ACTION A502_Suspending_Exit:
{attribute 'hide'}
IF NOT in_bDisableStateMethods THEN
	THIS^.M502_Suspending_Exit();
END_IF
END_ACTION

{attribute 'hide'}
METHOD M500_Suspending_Entry : BOOL
END_METHOD

{attribute 'hide'}
METHOD M501_Suspending : BOOL
VAR_OUTPUT
	(* Move to the Suspended state*)
	bSuspended	: BOOL	:= FALSE;
	(* Move to the Stopping state*)
	bStop		: BOOL	:= FALSE;
	(* Move to the Aborting state*)
	bAbort		: BOOL	:= FALSE;
END_VAR
// Go to suspended state by default
bSuspended := TRUE;
END_METHOD

{attribute 'hide'}
METHOD M502_Suspending_Exit : BOOL
END_METHOD

ACTION A510_Suspended_Entry:
{attribute 'hide'}
sm_enumState := E_PackMLState.Suspended;
sm_bUnsuspend := FALSE;

IF NOT in_bDisableStateMethods THEN
	THIS^.M_LogMessage('Entered $'Suspended$' state.');
	THIS^.M510_Suspended_Entry();
ELSE
	THIS^.M_LogWarning('State methods disabled! Entered $'Suspended$' state. Waiting for transition...');
END_IF
END_ACTION

ACTION A511_Suspended:
{attribute 'hide'}
IF NOT in_bDisableStateMethods THEN
	THIS^.M511_Suspended(
		bUnsuspend => sm_bUnsuspendCmd,
		bStop => sm_bStopCmd,
		bAbort => sm_bAbortCmd);
	IF sm_bAbortCmd THEN
		sm_bAbort := TRUE;
	ELSIF sm_bStopCmd THEN
		sm_bStop := TRUE;
	ELSIF sm_bUnsuspendCmd THEN
		sm_bUnsuspend := TRUE;
	END_IF
END_IF
END_ACTION

ACTION A512_Suspended_Exit:
{attribute 'hide'}
IF NOT in_bDisableStateMethods THEN
	THIS^.M512_Suspended_Exit();
END_IF
END_ACTION

{attribute 'hide'}
METHOD M510_Suspended_Entry : BOOL
END_METHOD

{attribute 'hide'}
METHOD M511_Suspended : BOOL
VAR_OUTPUT
	(* Move to the Unsuspending state*)
	bUnsuspend	: BOOL	:= FALSE;
	(* Move to the Stopping state*)
	bStop		: BOOL	:= FALSE;
	(* Move to the Aborting state*)
	bAbort		: BOOL	:= FALSE;
END_VAR
END_METHOD

{attribute 'hide'}
METHOD M512_Suspended_Exit : BOOL
END_METHOD

ACTION A520_Unsuspending_Entry:
{attribute 'hide'}
sm_enumState := E_PackMLState.Unsuspending;
sm_bUnsuspended := FALSE;

IF NOT in_bDisableStateMethods THEN
	THIS^.M_LogMessage('Entered $'Unsuspending$' state.');
	THIS^.M520_Unsuspending_Entry();
ELSE
	THIS^.M_LogWarning('State methods disabled! Entered $'Unsuspending$' state. Skipping to $'Execute$' state...');
	sm_bUnsuspended := TRUE;
END_IF
END_ACTION

ACTION A521_Unsuspending:
{attribute 'hide'}
IF NOT in_bDisableStateMethods THEN
	THIS^.M521_Unsuspending(
		bUnsuspended => sm_bUnsuspendedCmd,
		bStop => sm_bStopCmd,
		bAbort => sm_bAbortCmd);
	IF sm_bAbortCmd THEN
		sm_bAbort := TRUE;
	ELSIF sm_bStopCmd THEN
		sm_bStop := TRUE;
	ELSIF sm_bUnsuspendedCmd THEN
		sm_bUnsuspended := TRUE;
	END_IF
END_IF
END_ACTION

ACTION A522_Unsuspending_Exit:
{attribute 'hide'}
IF NOT in_bDisableStateMethods THEN
	THIS^.M522_Unsuspending_Exit();
END_IF
END_ACTION

{attribute 'hide'}
METHOD M520_Unsuspending_Entry : BOOL
END_METHOD

{attribute 'hide'}
METHOD M521_Unsuspending : BOOL
VAR_OUTPUT
	(* Move to the Execute state*)
	bUnsuspended	: BOOL	:= FALSE;
	(* Move to the Stopping state*)
	bStop			: BOOL	:= FALSE;
	(* Move to the Aborting state*)
	bAbort			: BOOL	:= FALSE;
END_VAR
// Move to the execute state by default
bUnsuspended := TRUE;
END_METHOD

{attribute 'hide'}
METHOD M522_Unsuspending_Exit : BOOL
END_METHOD

ACTION A_StateMachine:
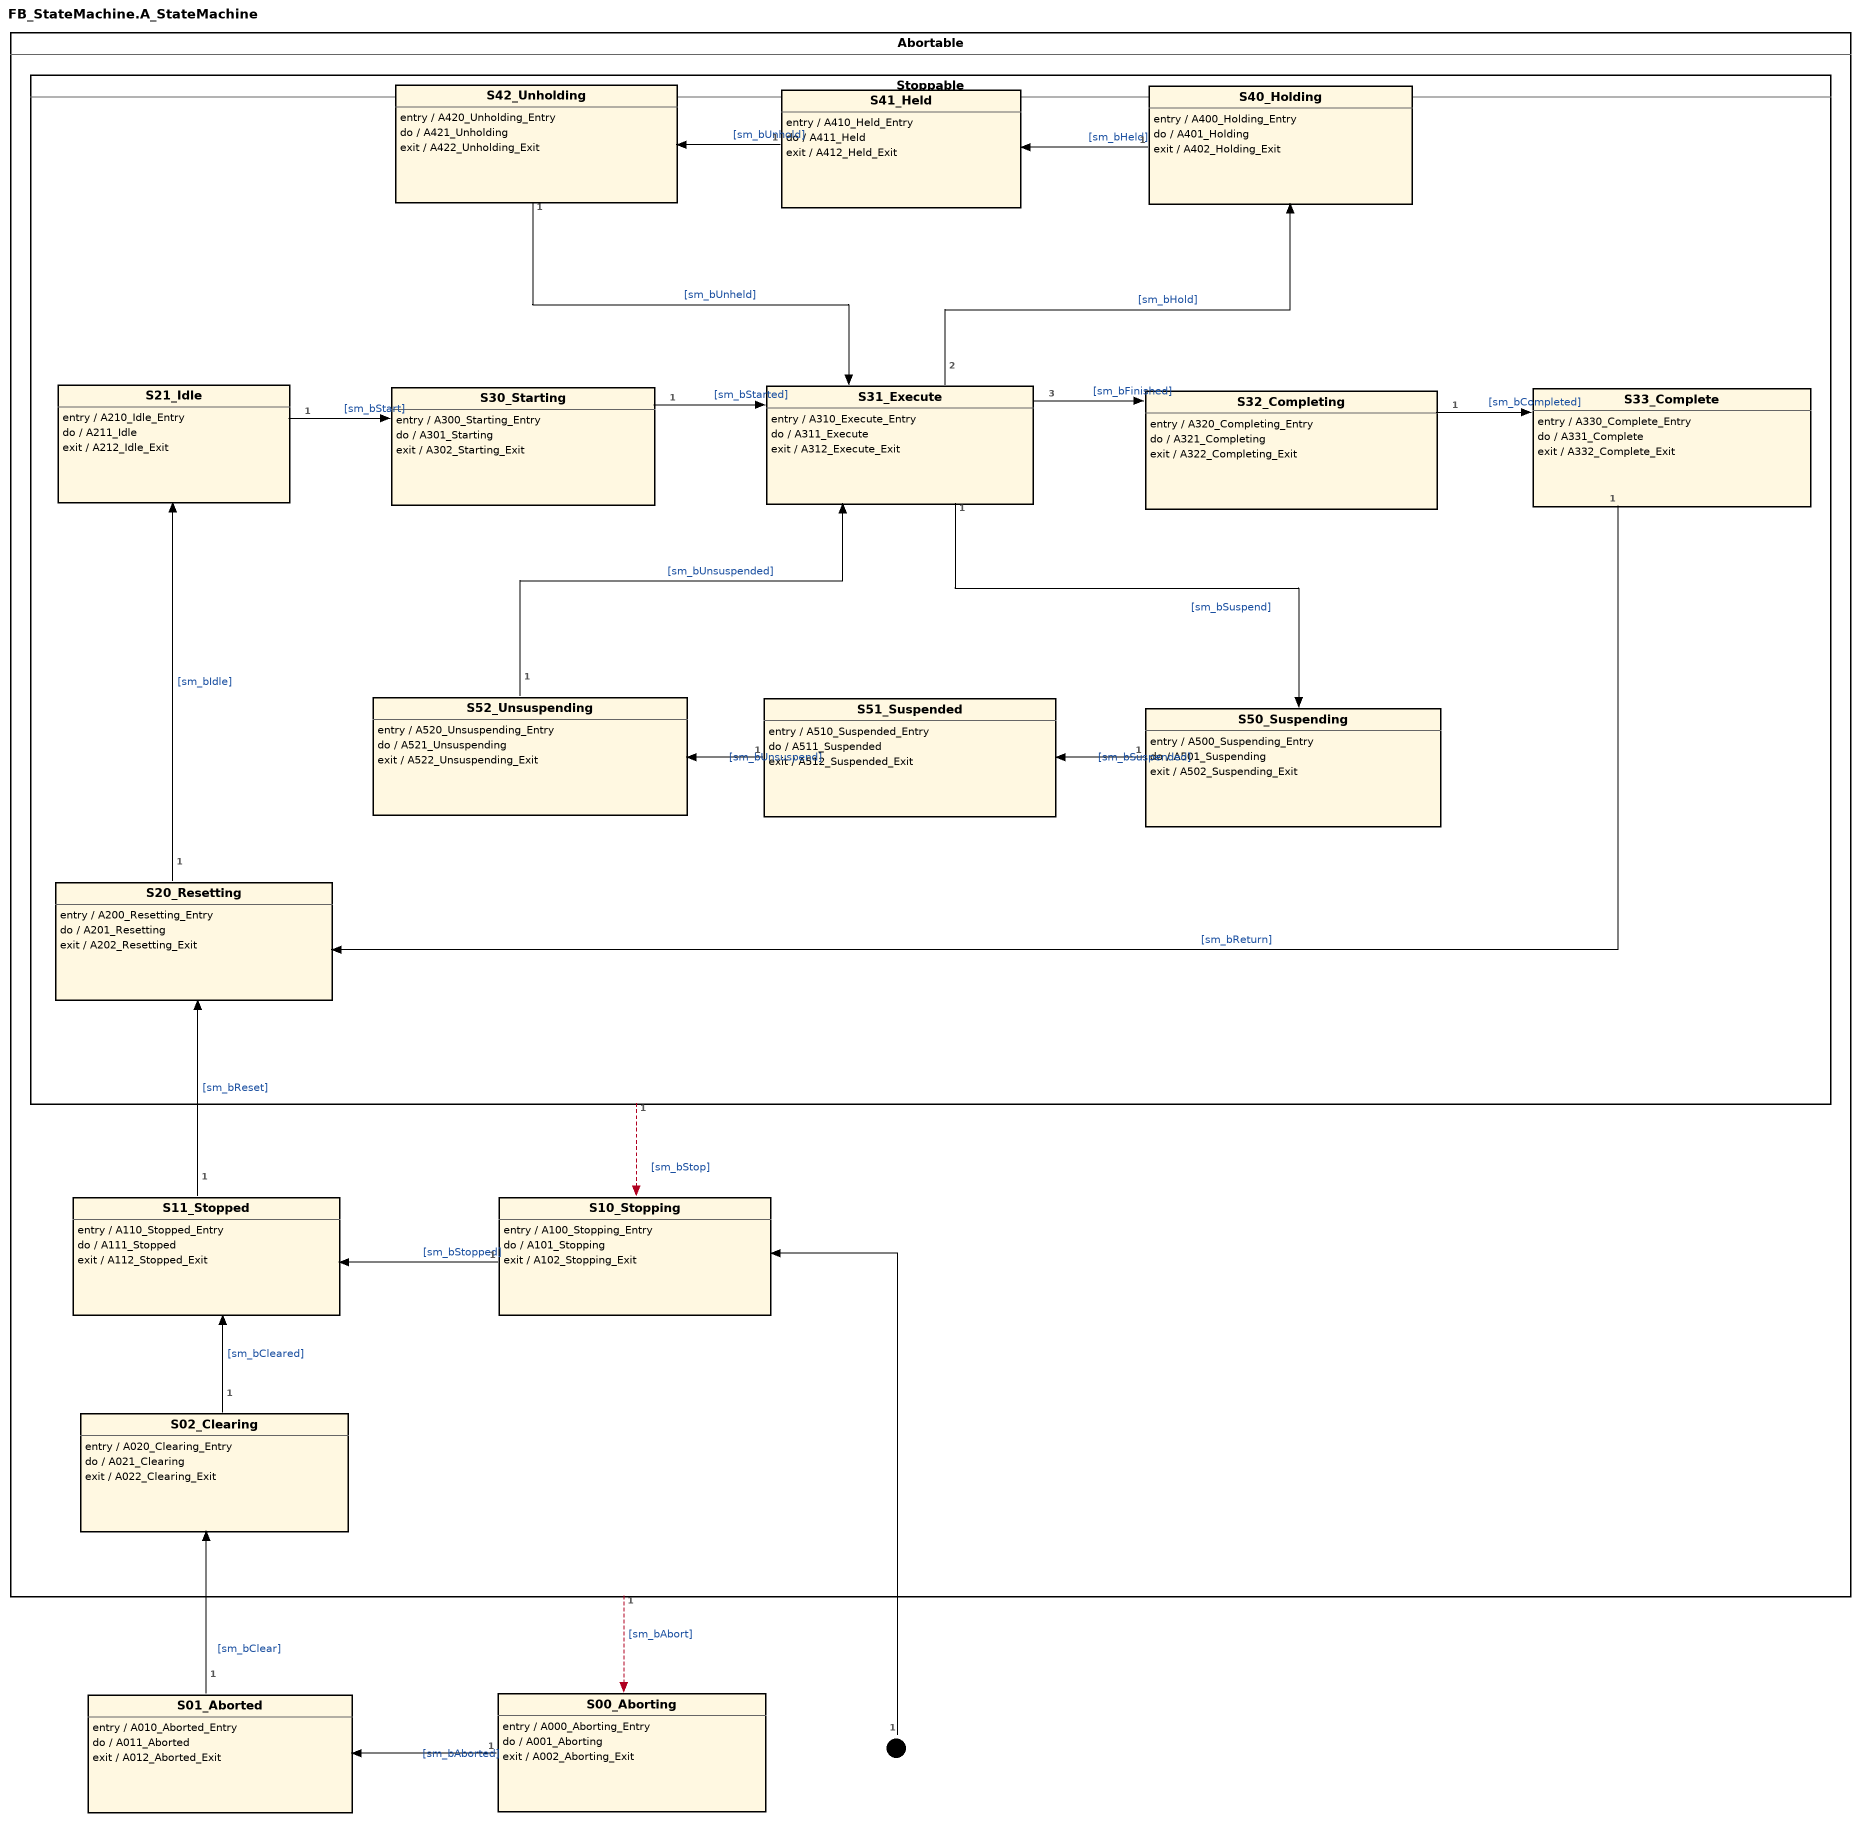
STATECHART A_StateMachine  // abortable
    START StartState1
    COMPOSITE STATE Abortable
        COMPOSITE STATE Stoppable
            STATE S42_Unholding
                entry / A420_Unholding_Entry
                do / A421_Unholding
                exit / A422_Unholding_Exit
            STATE S41_Held
                entry / A410_Held_Entry
                do / A411_Held
                exit / A412_Held_Exit
            STATE S40_Holding
                entry / A400_Holding_Entry
                do / A401_Holding
                exit / A402_Holding_Exit
            STATE S21_Idle
                entry / A210_Idle_Entry
                do / A211_Idle
                exit / A212_Idle_Exit
            STATE S30_Starting
                entry / A300_Starting_Entry
                do / A301_Starting
                exit / A302_Starting_Exit
            STATE S31_Execute
                entry / A310_Execute_Entry
                do / A311_Execute
                exit / A312_Execute_Exit
            STATE S32_Completing
                entry / A320_Completing_Entry
                do / A321_Completing
                exit / A322_Completing_Exit
            STATE S33_Complete
                entry / A330_Complete_Entry
                do / A331_Complete
                exit / A332_Complete_Exit
            STATE S52_Unsuspending
                entry / A520_Unsuspending_Entry
                do / A521_Unsuspending
                exit / A522_Unsuspending_Exit
            STATE S51_Suspended
                entry / A510_Suspended_Entry
                do / A511_Suspended
                exit / A512_Suspended_Exit
            STATE S50_Suspending
                entry / A500_Suspending_Entry
                do / A501_Suspending
                exit / A502_Suspending_Exit
            STATE S20_Resetting
                entry / A200_Resetting_Entry
                do / A201_Resetting
                exit / A202_Resetting_Exit
            S42_Unholding -> S31_Execute [sm_bUnheld] // priority 1
            S41_Held -> S42_Unholding [sm_bUnhold] // priority 1
            S40_Holding -> S41_Held [sm_bHeld] // priority 1
            S21_Idle -> S30_Starting [sm_bStart] // priority 1
            S30_Starting -> S31_Execute [sm_bStarted] // priority 1
            S31_Execute -> S50_Suspending [sm_bSuspend] // priority 1
            S31_Execute -> S40_Holding [sm_bHold] // priority 2
            S31_Execute -> S32_Completing [sm_bFinished] // priority 3
            S32_Completing -> S33_Complete [sm_bCompleted] // priority 1
            S33_Complete -> S20_Resetting [sm_bReturn] // priority 1
            S52_Unsuspending -> S31_Execute [sm_bUnsuspended] // priority 1
            S51_Suspended -> S52_Unsuspending [sm_bUnsuspend] // priority 1
            S50_Suspending -> S51_Suspended [sm_bSuspended] // priority 1
            S20_Resetting -> S21_Idle [sm_bIdle] // priority 1
        END_STATE
        STATE S11_Stopped
            entry / A110_Stopped_Entry
            do / A111_Stopped
            exit / A112_Stopped_Exit
        STATE S10_Stopping
            entry / A100_Stopping_Entry
            do / A101_Stopping
            exit / A102_Stopping_Exit
        STATE S02_Clearing
            entry / A020_Clearing_Entry
            do / A021_Clearing
            exit / A022_Clearing_Exit
        Stoppable -> S10_Stopping [sm_bStop] // priority 1, exception
        S11_Stopped -> S20_Resetting [sm_bReset] // priority 1
        S10_Stopping -> S11_Stopped [sm_bStopped] // priority 1
        S02_Clearing -> S11_Stopped [sm_bCleared] // priority 1
    END_STATE
    STATE S01_Aborted
        entry / A010_Aborted_Entry
        do / A011_Aborted
        exit / A012_Aborted_Exit
    STATE S00_Aborting
        entry / A000_Aborting_Entry
        do / A001_Aborting
        exit / A002_Aborting_Exit
    StartState1 -> S10_Stopping  // priority 1, on completion
    Abortable -> S00_Aborting [sm_bAbort] // priority 1, exception
    S01_Aborted -> S02_Clearing [sm_bClear] // priority 1
    S00_Aborting -> S01_Aborted [sm_bAborted] // priority 1
END_STATECHART
END_ACTION

END_FUNCTION_BLOCK

// Interfaces/State Machine/I_StateControl
(* The state control interface should be implemented on stateful modules that
cannot move on from wait states automatically due to being controlled by
external modules. *)
INTERFACE I_StateControl

(* Go to the aborting state while in the stoppable or abortable group. *)
METHOD M_Abort : BOOL
VAR_INPUT
END_VAR
END_METHOD

(* Go to the clearing state from the aborted state. *)
METHOD M_Clear : BOOL
VAR_INPUT
END_VAR
END_METHOD

(* Go to the completing state from the execute state. *)
METHOD M_Complete : BOOL
VAR_INPUT
END_VAR
END_METHOD

(* Go to the holding state from the execute state. *)
METHOD M_Hold : BOOL
VAR_INPUT
END_VAR
END_METHOD

(* Go to the resetting state from the stopped state. *)
METHOD M_Reset : BOOL
VAR_INPUT
END_VAR
END_METHOD

(* Go to the resetting state from the complete state. *)
METHOD M_Return : BOOL
VAR_INPUT
END_VAR
END_METHOD

(* Go to the execute state from the idle state. *)
METHOD M_Start : BOOL
VAR_INPUT
END_VAR
END_METHOD

(* Go to the stopping state while in the stoppable group. *)
METHOD M_Stop : BOOL
VAR_INPUT
END_VAR
END_METHOD

(* Go to the suspending state from the execute state. *)
METHOD M_Suspend : BOOL
VAR_INPUT
END_VAR
END_METHOD

(* Go to the unholding state from the held state. *)
METHOD M_Unhold : BOOL
VAR_INPUT
END_VAR
END_METHOD

(* Go to the unsuspending state from the suspended state. *)
METHOD M_Unsuspend : BOOL
VAR_INPUT
END_VAR
END_METHOD

END_INTERFACE

// Interfaces/Machines/I_MachineStationStateControl
INTERFACE I_MachineStationStateControl

(* Executes M_Abort on all stations and returns TRUE when M_Abort
	returns TRUE on all stations. *)
METHOD M_AbortStations : BOOL
VAR_INPUT
END_VAR
END_METHOD

(* Executes M_Clear on all stations and returns TRUE when M_Clear
	returns TRUE on all stations. *)
METHOD M_ClearStations : BOOL
VAR_INPUT
END_VAR
END_METHOD

(* Executes M_Complete on all stations and returns TRUE when M_Complete
	returns TRUE on all stations. *)
METHOD M_CompleteStations : BOOL
VAR_INPUT
END_VAR
END_METHOD

(* Executes M_Hold on all stations and returns TRUE when M_Hold 
	returns TRUE on all stations. *)
METHOD M_HoldStations : BOOL
VAR_INPUT
END_VAR
END_METHOD

(* Executes M_Reset on all stations and returns TRUE when M_Reset 
	returns TRUE on all stations. *)
METHOD M_ResetStations : BOOL
VAR_INPUT
END_VAR
END_METHOD

(* Executes M_Return on all stations and returns TRUE when M_Return 
	returns TRUE on all stations. *)
METHOD M_ReturnStations : BOOL
VAR_INPUT
END_VAR
END_METHOD

(* Executes M_Start on all stations and returns TRUE when M_Start 
	returns TRUE on all stations. *)
METHOD M_StartStations : BOOL
VAR_INPUT
END_VAR
END_METHOD

(* Executes M_Stop on all stations and returns TRUE when M_Stop 
	returns TRUE on all stations. *)
METHOD M_StopStations : BOOL
VAR_INPUT
END_VAR
END_METHOD

(* Executes M_Suspend on all stations and returns TRUE when M_Suspend
	returns TRUE on all stations. *)
METHOD M_SuspendStations : BOOL
VAR_INPUT
END_VAR
END_METHOD

(* Executes M_Unhold on all stations and returns TRUE when M_Unhold
	returns TRUE on all stations. *)
METHOD M_UnholdStations : BOOL
VAR_INPUT
END_VAR
END_METHOD

(* Executes M_Unsuspend on all stations and returns TRUE when M_Unsuspend
	returns TRUE on all stations. *)
METHOD M_UnsuspendStations : BOOL
VAR_INPUT
END_VAR
END_METHOD

END_INTERFACE

// Abstract/FB_Station
(*
===============================================================================
Station
===============================================================================
:Contact: Kevin Sanita <ksanita@sensata.com>
:Last Edited: March 2022

:Description: Represents a station, which is a collection of devices that interact with each other.

:Notes:
* Stations are able to implement state machines. To implement a state machine, implement I_Stateful
* In order for a state machine to run, THIS^.A_StateMachine must be called in the function block body.

:Change Log:
- **December 2021** Initial version
- **March 16, 2022** Added device list controls
*)
{attribute 'hide_all_locals'}
FUNCTION_BLOCK ABSTRACT FB_Station EXTENDS FB_StateMachine IMPLEMENTS I_StationDeviceControl
VAR_INPUT
END_VAR
VAR_OUTPUT
END_VAR
VAR
	sta_arrDevices : T_StationDeviceArray;
END_VAR

(* Calls the abort method on all devices in a station. *)
METHOD M_AbortDevices : BOOL

VAR
	uintIndex: UINT;
	fbDevice : POINTER TO FB_Device;
	bDeviceAborted: BOOL;
END_VAR
// Initialize result to true
M_AbortDevices := TRUE;

// Run through each device
FOR uintIndex := 1 TO GVL_Constants.uintMAX_STATION_DEVICE_COUNT DO
	// If the pointer is set
	IF sta_arrDevices[uintIndex] > 0 THEN
		// Get the device from the pointer
		fbDevice := sta_arrDevices[uintIndex];
		
		// Abort the device
		bDeviceAborted := fbDevice^.M_Abort();
		
		// If the abort is not finished, return false
		IF NOT bDeviceAborted THEN
			M_AbortDevices := FALSE;
		END_IF
	END_IF
END_FOR
END_METHOD

(* Calls the connect method on all devices in a station. *)
METHOD M_ConnectDevices : BOOL

VAR
	uintIndex: UINT;
	fbDevice: POINTER TO FB_Device;
	bDeviceConnected: BOOL;
END_VAR
// Initialize result to true
M_ConnectDevices := TRUE;

// Run through each device
FOR uintIndex := 1 TO GVL_Constants.uintMAX_STATION_DEVICE_COUNT DO
	// If the pointer is set
	IF sta_arrDevices[uintIndex] > 0 THEN
		// Get the device from the pointer
		fbDevice := sta_arrDevices[uintIndex];
		
		// Try to connect
		bDeviceConnected := fbDevice^.M_Connect();
		
		// If not connected, return false
		IF NOT bDeviceConnected THEN
			M_ConnectDevices := FALSE;
		END_IF
		
	END_IF
END_FOR
END_METHOD

(* Calls the disable method on all devices in a station. *)
METHOD M_DisableDevices : BOOL

VAR
	uintIndex: UINT;
	fbDevice: POINTER TO FB_Device;
	bDeviceDisabled: BOOL;
END_VAR
// Initialize result to True
M_DisableDevices := TRUE;

// Run through each device
FOR uintIndex := 1 TO GVL_Constants.uintMAX_STATION_DEVICE_COUNT DO
	// If the pointer is set
	IF sta_arrDevices[uintIndex] > 0 THEN
		// Get the device from the pointer
		fbDevice := sta_arrDevices[uintIndex];
		
		// Try to disable device
		bDeviceDisabled := fbDevice^.M_Disable();
		
		// Return false if the device is not disabled
		IF NOT bDeviceDisabled THEN
			M_DisableDevices := FALSE;
		END_IF
		
	END_IF
END_FOR
END_METHOD

(* Calls the disconnect method on all devices in a station. *)
METHOD M_DisconnectDevices : BOOL

VAR
	uintIndex: UINT;
	fbDevice: POINTER TO FB_Device;
	bDeviceDisconnected: BOOL;
END_VAR
M_DisconnectDevices := TRUE;

// Run through each device
FOR uintIndex := 1 TO GVL_Constants.uintMAX_STATION_DEVICE_COUNT DO
	// If the pointer is set
	IF sta_arrDevices[uintIndex] > 0 THEN
		// Get the device from the pointer
		fbDevice := sta_arrDevices[uintIndex];
		
		// Try to disconnect the device
		bDeviceDisconnected := fbDevice^.M_Disconnect();
		
		// If the device is not disconnected, return false
		IF NOT bDeviceDisconnected THEN
			M_DisconnectDevices := FALSE;
		END_IF
		
	END_IF
END_FOR
END_METHOD

(*
Checks for errors on all devices in the station
*)
METHOD M_ElevateDeviceErrors : BOOL
VAR_INPUT
END_VAR

VAR
	uintIndex: UINT;
	fbDevice: POINTER TO FB_Device;
	udintErrorNo: UDINT;
	strErrorDescription: T_MaxString;
END_VAR
M_ElevateDeviceErrors := FALSE;

// Run through each device
FOR uintIndex := 1 TO GVL_Constants.uintMAX_STATION_DEVICE_COUNT DO
	// If the pointer is set
	IF sta_arrDevices[uintIndex] > 0 THEN
		// Get the device from the pointer
		fbDevice := sta_arrDevices[uintIndex];
		
		// Check device for error and set error if there is one
		IF fbDevice^.P_bError THEN
			udintErrorNo := E_StationError.DeviceError;
			udintErrorNo := udintErrorNo + uintIndex;
			strErrorDescription := CONCAT('Device ', fbDevice^.in_strUniqueId);
			strErrorDescription := CONCAT(strErrorDescription, 'has the following error: ');
			strErrorDescription := CONCAT(strErrorDescription, fbDevice^.P_strErrorMessage);
			
			THIS^.M_SetError(
				udintErrorNo,
				strErrorDescription);
				
			M_ElevateDeviceErrors := TRUE;
		END_IF
	END_IF
END_FOR
END_METHOD

(* Calls the enable method on all devices in a station. *)
METHOD M_EnableDevices : BOOL

VAR
	uintIndex: UINT;
	fbDevice: POINTER TO FB_Device;
	bDeviceEnabled: BOOL;
END_VAR
M_EnableDevices := TRUE;

// Run through each device
FOR uintIndex := 1 TO GVL_Constants.uintMAX_STATION_DEVICE_COUNT DO
	// If the pointer is set
	IF sta_arrDevices[uintIndex] > 0 THEN
		// Get the device from the pointer
		fbDevice := sta_arrDevices[uintIndex];
		
		// Try to enable the device
		bDeviceEnabled := fbDevice^.M_Enable();
		
		// If the device is not enabled, return false
		IF NOT bDeviceEnabled THEN
			M_EnableDevices := FALSE;
		END_IF
		
	END_IF
END_FOR
END_METHOD

(* Calls the pause method on all devices in a station. *)
METHOD M_PauseDevices : BOOL

VAR
	uintIndex: UINT;
	fbDevice: POINTER TO FB_Device;
	bDevicePaused: BOOL;
END_VAR
M_PauseDevices := TRUE;

// Run through each device
FOR uintIndex := 1 TO GVL_Constants.uintMAX_STATION_DEVICE_COUNT DO
	// If the pointer is set
	IF sta_arrDevices[uintIndex] > 0 THEN
		// Get the device from the pointer
		fbDevice := sta_arrDevices[uintIndex];
		
		// Try to pause the device
		bDevicePaused := fbDevice^.M_PauseProgram();
		
		// If the device is not paused, return false
		IF NOT bDevicePaused THEN
			M_PauseDevices := FALSE;
		END_IF

	END_IF
END_FOR
END_METHOD

(* Calls the power off method on all devices in a station. *)
METHOD M_PowerOffDevices : BOOL

VAR
	uintIndex: UINT;
	fbDevice: POINTER TO FB_Device;
	bDeviceOff: BOOL;
END_VAR
M_PowerOffDevices := TRUE;

// Run through each device
FOR uintIndex := 1 TO GVL_Constants.uintMAX_STATION_DEVICE_COUNT DO
	// If the pointer is set
	IF sta_arrDevices[uintIndex] > 0 THEN
		// Get the device from the pointer
		fbDevice := sta_arrDevices[uintIndex];
		
		// Try to power off the device
		bDeviceOff := fbDevice^.M_PowerOff();
		
		// If the device is not powered off, return false
		IF NOT bDeviceOff THEN
			M_PowerOffDevices := FALSE;
		END_IF
		
	END_IF
END_FOR
END_METHOD

(* Calls the power on method on all devices in a station. *)
METHOD M_PowerOnDevices : BOOL

VAR
	uintIndex: UINT;
	fbDevice: POINTER TO FB_Device;
	bDeviceOn: BOOL;
END_VAR
M_PowerOnDevices := TRUE;

// Run through each device
FOR uintIndex := 1 TO GVL_Constants.uintMAX_STATION_DEVICE_COUNT DO
	// If the pointer is set
	IF sta_arrDevices[uintIndex] > 0 THEN
		// Get the device from the pointer
		fbDevice := sta_arrDevices[uintIndex];
		
		// Try to power on device
		bDeviceOn := fbDevice^.M_PowerOn();
		
		// If the device is not on, return false
		IF NOT bDeviceOn THEN
			M_PowerOnDevices := FALSE;
		END_IF
		
	END_IF
END_FOR
END_METHOD

(* Calls the reset method on all devices in a station. *)
METHOD M_ResetDevices : BOOL

VAR
	uintIndex: UINT;
	fbDevice: POINTER TO FB_Device;
	bDeviceReset: BOOL;
END_VAR
M_ResetDevices := TRUE;

// Run through each device
FOR uintIndex := 1 TO GVL_Constants.uintMAX_STATION_DEVICE_COUNT DO
	// If the pointer is set
	IF sta_arrDevices[uintIndex] > 0 THEN
		// Get the device from the pointer
		fbDevice := sta_arrDevices[uintIndex];
		
		// Try to reset the device
		bDeviceReset := fbDevice^.M_Reset();
		
		// If device is not reset, return false
		IF NOT bDeviceReset THEN
			M_ResetDevices := FALSE;
		END_IF
		
	END_IF
END_FOR
END_METHOD

(* Calls the start method on all devices in a station. *)
METHOD M_StartDevices : BOOL

VAR
	uintIndex: UINT;
	fbDevice: POINTER TO FB_Device;
	bDeviceStarted: BOOL;
END_VAR
M_StartDevices := TRUE;

// Run through each device
FOR uintIndex := 1 TO GVL_Constants.uintMAX_STATION_DEVICE_COUNT DO
	// If the pointer is set
	IF sta_arrDevices[uintIndex] > 0 THEN
		// Get the device from the pointer
		fbDevice := sta_arrDevices[uintIndex];
		
		bDeviceStarted := fbDevice^.M_StartProgram();
		
		IF NOT bDeviceStarted THEN
			M_StartDevices := FALSE;
		END_IF
	END_IF
END_FOR
END_METHOD

(* Calls the stop method on all devices in a station. *)
METHOD M_StopDevices : BOOL

VAR
	uintIndex: UINT;
	fbDevice: POINTER TO FB_Device;
	bDeviceStopped: BOOL;
END_VAR
M_StopDevices := TRUE;

// Run through each device
FOR uintIndex := 1 TO GVL_Constants.uintMAX_STATION_DEVICE_COUNT DO
	// If the pointer is set
	IF sta_arrDevices[uintIndex] > 0 THEN
		// Get the device from the pointer
		fbDevice := sta_arrDevices[uintIndex];
		
		// Try to stop the device
		bDeviceStopped := fbDevice^.M_StopProgram();
		
		// If the device is not stopped, return false
		IF NOT bDeviceStopped THEN
			M_StopDevices := FALSE;
		END_IF
		
	END_IF
END_FOR
END_METHOD

(* Adds a device to the device list. *)
METHOD M_SetDevice : BOOL
VAR_INPUT
	(* Index of device to set. Between 1 and uintMAX_STATION_DEVICE_COUNT. *)
	uintIndex : UINT;
	
	(* Reference to the device to add to the device array. *)
	refDevice : REFERENCE TO FB_Device;
	
END_VAR
IF uintIndex > 0 AND uintIndex <= GVL_Constants.uintMAX_STATION_DEVICE_COUNT THEN
	sta_arrDevices[uintIndex] := ADR(refDevice);
	M_SetDevice := TRUE;
ELSE
	M_SetDevice := FALSE;
END_IF
END_METHOD

(* The array of device pointers for this station. *)
PROPERTY P_arrDevices : T_StationDeviceArray
GET
P_arrDevices := sta_arrDevices;
END_GET
END_PROPERTY

END_FUNCTION_BLOCK

// Interfaces/Stations/I_StationDeviceControl
INTERFACE I_StationDeviceControl

(* Calls the abort method on all devices in a station. *)
METHOD M_AbortDevices : BOOL
VAR_INPUT
END_VAR
END_METHOD

(* Calls the connect method on all devices in a station. *)
METHOD M_ConnectDevices : BOOL
VAR_INPUT
END_VAR
END_METHOD

(* Calls the disconnect method on all devices in a station. *)
METHOD M_DisconnectDevices : BOOL
VAR_INPUT
END_VAR
END_METHOD

(* Calls the pause method on all devices in a station. *)
METHOD M_PauseDevices : BOOL
VAR_INPUT
END_VAR
END_METHOD

(* Calls the start method on all devices in a station. *)
METHOD M_StartDevices : BOOL
VAR_INPUT
END_VAR
END_METHOD

(* Calls the stop method on all devices in a station. *)
METHOD M_StopDevices : BOOL
VAR_INPUT
END_VAR
END_METHOD

(* Calls the disable method on all devices in a station. *)
METHOD M_DisableDevices : BOOL
VAR_INPUT
END_VAR
END_METHOD

(* Calls the enable method on all devices in a station. *)
METHOD M_EnableDevices : BOOL
VAR_INPUT
END_VAR
END_METHOD

(* Calls the power off method on all devices in a station. *)
METHOD M_PowerOffDevices : BOOL
VAR_INPUT
END_VAR
END_METHOD

(* Calls the power on method on all devices in a station. *)
METHOD M_PowerOnDevices : BOOL
VAR_INPUT
END_VAR
END_METHOD

(* Calls the reset method on all devices in a station. *)
METHOD M_ResetDevices : BOOL
VAR_INPUT
END_VAR
END_METHOD

(* Check all devices in the device list for errors. *)
METHOD M_ElevateDeviceErrors : BOOL
VAR_INPUT
END_VAR
END_METHOD

END_INTERFACE

// Concrete/FB_DeviceTestStation
FUNCTION_BLOCK FB_DeviceTestStation EXTENDS FB_Station IMPLEMENTS I_Stateful
VAR_INPUT
	ref_fbDevice: REFERENCE TO FB_Device; // The device to be tested
	
	in_bAbortBtn: BOOL; // Abort from any abortable states
	in_bClearBtn: BOOL; // Clear the abort state and any errors
	in_bStopBtn: BOOL; // Stop from any stoppable states
	in_bResetBtn: BOOL; // Return to the idle state from stopped or completed
	in_bStartBtn: BOOL; // Start from idle or restart from held or suspended
	in_bCompleteBtn: BOOL; // Exit the execute step to the complete step
	in_bHoldBtn: BOOL; // Hold the machine while in execute state
	in_bSuspendBtn: BOOL; // Suspend the machine while in execute state
	
	in_strProgram: T_MaxString; // Program to load when testing program loading
END_VAR
VAR_OUTPUT
	out_bAbortTested: BOOL; // Gets set to TRUE once M_Abort on ref_fbDevice has been tested once
	
	out_bConnectTested: BOOL;  // Gets set to TRUE once M_Connect on ref_fbDevice has been tested once
	out_bDisconnectTested: BOOL;  // Gets set to TRUE once M_Disconnect on ref_fbDevice has been tested once
	
	out_bEnableTested: BOOL; // Gets set to TRUE once M_Enable on ref_fbDevice has been tested once
	out_bDisableTested: BOOL; // Gets set to TRUE once M_Disable on ref_fbDevice has been tested once
	
	out_bPowerOnTested: BOOL; // Gets set to TRUE once M_PowerOn on ref_fbDevice has been tested once
	out_bPowerOffTested: BOOL; // Gets set to TRUE once M_PowerOff on ref_fbDevice has been tested once
	
	out_bLoadProgramTested: BOOL; // Gets set to TRUE once M_LoadProgram on ref_fbDevice has been tested once
	out_bStartProgramTested: BOOL; // Gets set to TRUE once M_StartProgram on ref_fbDevice has been tested once
	out_bStopProgramTested: BOOL; // Gets set to TRUE once M_StopProgram on ref_fbDevice has been tested once
	out_bPauseProgramTested: BOOL; // Gets set to TRUE once M_PauseProgram on ref_fbDevice has been tested once
	out_bUnpauseProgramTested: BOOL; // Gets set to TRUE once M_StartProgram on ref_fbDevice has been tested once after M_PauseProgram was used
	out_bStopPausedProgramTested: BOOL; // Gets set to TRUE once M_StopProgram on ref_fbDevice has been tested once after M_PauseProgram was used
	
	out_bResetTested: BOOL; // Gets set to TRUE once M_Reset on ref_fbDevice has been tested once
END_VAR
VAR
	bDeviceReset: BOOL;
	
	bDeviceConnected: BOOL;
	bDeviceDisconnected: BOOL;
	
	bDevicePoweredOn: BOOL;
	bDevicePoweredOff: BOOL;
	
	bDeviceEnabled: BOOL;
	bDeviceDisabled: BOOL;
	
	bDeviceProgramLoaded: BOOL;
	bDeviceProgramStarted: BOOL;
	bDeviceProgramStopped: BOOL;
	bDeviceProgramPaused: BOOL;

	// Device test trackers
	fbDeviceAborted: R_TRIG;
	fbDeviceReset: F_TRIG;
	fbDeviceConnected: R_TRIG;
	fbDeviceDisconnected: F_TRIG;
	fbDeviceEnabled: R_TRIG;
	fbDeviceDisabled: F_TRIG;
	fbDevicePoweredOn: R_TRIG;
	fbDevicePoweredOff: F_TRIG;
	fbDeviceProgramLoaded: R_TRIG;
	enumLastState: E_ProgramState;
END_VAR

THIS^.M_SetDevice(1, ref_fbDevice);

A_StateMachine();

A_DeviceTestTracking();

(* Runs for a single cycle when entering the aborting state. *)
METHOD M000_Aborting_Entry : BOOL
THIS^.M_LogMessage('Aborting');
END_METHOD

(* The 'Aborting' state can be entered at any time while within the 'abortable'
section of the state machine. It is typically entered in response to an 'Abort'
command or a critical fault. The logic should safely but rapidly bring the
components of the module to a stop while maintaining as much information about
the pre-abort scenario as possible. *)
METHOD M001_Aborting : BOOL
VAR_OUTPUT
	(* This should be set to true once all components of the module have safely
	come to a stop. Once set to true, the state machine will move to the
	'Aborted' state. *)
	bAborted	: BOOL;
END_VAR
// Go to the aborted state once the device is aborted
bAborted := ref_fbDevice.M_Abort();
END_METHOD

(* Runs for a single cycle when exiting the aborting state. *)
METHOD M002_Aborting_Exit : BOOL
END_METHOD

(* Runs for a single cycle when entering the aborted state. *)
METHOD M010_Aborted_Entry : BOOL
THIS^.M_LogMessage('Aborted');
END_METHOD

(* This state is entered after the aborting state completes, and should
not modify anything in the module while awaiting an explicit 'Clear' command. *)
METHOD M011_Aborted : BOOL
VAR_OUTPUT
	(* This should be set to true once an explicit 'Clear' command is received.
	Once set to true, the state machine will move to the 'Clearing' state. *)
	bClear	: BOOL;
END_VAR
// Only go to clearing state if clear button is pressed
bClear := in_bClearBtn;
END_METHOD

(* Runs for a single cycle when exiting the aborted state. *)
METHOD M012_Aborted_Exit : BOOL
END_METHOD

(* Runs for a single cycle when entering the clearing state. *)
METHOD M020_Clearing_Entry : BOOL
THIS^.M_LogMessage('Clearing');
END_METHOD

(* This state should clear any faults and reset any safety features related
to the module, as well as perform actions similar to the 'Stopping' state
if they were not already performed while aborting. *)
METHOD M021_Clearing : BOOL
VAR_OUTPUT
	(* This should be set to true once the safety state of all module
	components are reset and all errors are cleared. *)
	bCleared	: BOOL;
	(* This should be set to true if a potentially hazardous error or a safety
	fault has occurred in any tasks. Once set to true, the state machine will
	move to the 'Aborting' state. *)
	bAbort	: BOOL;
END_VAR
// Exit once the device is reset
bCleared := ref_fbDevice.M_Reset();

// If device is reset, clear module errors
IF bCleared THEN
	THIS^.M_ClearError();
END_IF

// If the device has an error, abort
IF ref_fbDevice.P_bError THEN
	THIS^.M_SetError(200, 'Error on fbDevice!');
	bAbort := TRUE;
	
// Abort if abort button is pressed
ELSIF in_bAbortBtn THEN
	THIS^.M_SetError(100, 'Abort button pressed!');
	bAbort := TRUE;
END_IF
END_METHOD

(* Runs for a single cycle when exiting the clearing state. *)
METHOD M022_Clearing_Exit : BOOL
END_METHOD

(* Runs for a single cycle when entering the stopping state. *)
METHOD M100_Stopping_Entry : BOOL
THIS^.M_LogMessage('Stopping');

// Reset device status variables
bDeviceProgramStopped := FALSE;
bDeviceDisabled := FALSE;
bDevicePoweredOff := FALSE;
END_METHOD

(* This state can be entered from anywhere within the 'stoppable' group of
states. This state should safely bring the components of the module to a
controlled stop and then move to the 'Stopped' state once completed. *)
METHOD M101_Stopping : BOOL
VAR_OUTPUT
	(* This should be set to true once all relevant components have come to a
	controlled stop. Once set to true, the state machine will move to the
	'Stopped' state. *)
	bStopped	: BOOL;
	(* This should be set to true if a potentially hazardous error or a safety
	fault has occurred in any tasks. Once set to true, the state machine will
	move to the 'Aborting' state. *)
	bAbort	: BOOL;
END_VAR
// If the device is connected, stop and disable it
IF ref_fbDevice.P_bConnected THEN
	
	// Stop the program
	IF NOT bDeviceProgramStopped THEN
		bDeviceProgramStopped := ref_fbDevice.M_StopProgram();
		
	// Disable the device
	ELSIF NOT bDeviceDisabled THEN
		bDeviceDisabled := ref_fbDevice.M_Disable();
	
	// Power off the device
	ELSIF NOT bDevicePoweredOff THEN
		bDevicePoweredOff := ref_fbDevice.M_PowerOff();
		
	// Exit once stopped and disabled
	ELSE
		bStopped := TRUE;
	END_IF
	
// If the device is not connected, it can be considered to be stopped
ELSE
	bStopped := TRUE;
END_IF

// If the device has an error, abort
IF ref_fbDevice.P_bError THEN
	THIS^.M_SetError(200, 'Error on fbDevice!');
	bAbort := TRUE;
	
// Abort if abort button is pressed
ELSIF in_bAbortBtn THEN
	THIS^.M_SetError(100, 'Abort button pressed!');
	bAbort := TRUE;
END_IF
END_METHOD

(* Runs for a single cycle when exiting the stopping state. *)
METHOD M102_Stopping_Exit : BOOL
END_METHOD

(* Runs for a single cycle when entering the stopped state. *)
METHOD M110_Stopped_Entry : BOOL
THIS^.M_LogMessage('Stopped');
END_METHOD

(* The machine should be stationary and awaiting an explicit 'Reset' command
while in this state. Once the 'Reset' command is received, the state machine
will move to the 'Resetting' state. *)
METHOD M111_Stopped : BOOL
VAR_OUTPUT
	(* This should be set to true if an explicit reset command is received.
	Once set to true, the state machine will move to the 'Resetting' state. *)
	bReset	: BOOL;
	(* This should be set to true if a potentially hazardous error or a safety
	fault has occurred in any tasks. Once set to true, the state machine will
	move to the 'Aborting' state. *)
	bAbort	: BOOL;
END_VAR
// Go to the resetting state if the reset button is pressed
bReset := in_bResetBtn;

// If the device has an error, abort
IF ref_fbDevice.P_bError THEN
	THIS^.M_SetError(200, 'Error on fbDevice!');
	bAbort := TRUE;
	
// Abort if abort button is pressed
ELSIF in_bAbortBtn THEN
	THIS^.M_SetError(100, 'Abort button pressed!');
	bAbort := TRUE;
END_IF
END_METHOD

(* Runs for a single cycle when exiting the stopped state. *)
METHOD M112_Stopped_Exit : BOOL
END_METHOD

(* Runs for a single cycle when entering the resetting state. *)
METHOD M200_Resetting_Entry : BOOL
THIS^.M_LogMessage('Resetting');

// Reset device status variables
bDeviceDisconnected := FALSE;
bDeviceConnected := FALSE;
bDeviceReset := FALSE;
END_METHOD

(* This state should place the module and all of its components into a safe
energized idle state where it will wait for a start command. Once all tasks are
complete, it will move to the 'Idle' state. No external movement should occur
as a result of this state. *)
METHOD M201_Resetting : BOOL
VAR_OUTPUT
	(* Set this to true once the module is energized and ready to start.
	Once set to true, the state machine will move to the 'Idle' state. *)
	bIdle	: BOOL;
	(* This should be set to true if an external source requests that the module
	exit its current state and come to a controlled stop. Once set to true, the
	state machine will move to the 'Stopping' state. *)
	bStop	: BOOL;
	(* This should be set to true if a potentially hazardous error or a safety
	fault has occurred in any tasks. Once set to true, the state machine will
	move to the 'Aborting' state. *)
	bAbort	: BOOL;
END_VAR
// Stop if stop button is pressed
bStop := in_bStopBtn;

// Disconnect the device to reset the connection
IF NOT bDeviceDisconnected THEN
	bDeviceDisconnected := ref_fbDevice.M_Disconnect();
	
// Connect (or reconnect) the device
ELSIF NOT bDeviceConnected THEN
	bDeviceConnected := ref_fbDevice.M_Connect();
	
// Reset the device
ELSIF NOT bDeviceReset THEN
	bDeviceReset := ref_fbDevice.M_Reset();

// Once reconnected and reset, go to the idle state
ELSE
	bIdle := TRUE;
END_IF

// If the device has an error, abort
IF ref_fbDevice.P_bError THEN
	THIS^.M_SetError(200, 'Error on fbDevice!');
	bAbort := TRUE;
	
// Abort if abort button is pressed
ELSIF in_bAbortBtn THEN
	THIS^.M_SetError(100, 'Abort button pressed!');
	bAbort := TRUE;

END_IF
END_METHOD

(* Runs for a single cycle when exiting the resetting state. *)
METHOD M202_Resetting_Exit : BOOL
END_METHOD

(* Runs for a single cycle when entering the idle state. *)
METHOD M210_Idle_Entry : BOOL
THIS^.M_LogMessage('Idle');
END_METHOD

(* This state should maintain the status of the module and its components that
was set by the resetting step while awaiting an explicit 'Start' command. *)
METHOD M211_Idle : BOOL
VAR_OUTPUT
	(* This should be set to true if an explicit 'Start' command is received.
	Once set to true, the state machine will move to the 'Starting' state. *)
	bStart	: BOOL;
	(* This should be set to true if an external source requests that the module
	exit its current state and come to a controlled stop. Once set to true, the
	state machine will move to the 'Stopping' state. *)
	bStop	: BOOL;
	(* This should be set to true if a potentially hazardous error or a safety
	fault has occurred in any tasks. Once set to true, the state machine will
	move to the 'Aborting' state. *)
	bAbort	: BOOL;
END_VAR
// Start if start button is pressed
bStart := in_bStartBtn;

// Stop if stop button is pressed
bStop := in_bStopBtn;

// If the device has an error, abort
IF ref_fbDevice.P_bError THEN
	THIS^.M_SetError(200, 'Error on fbDevice!');
	bAbort := TRUE;
	
// Abort if abort button is pressed
ELSIF in_bAbortBtn THEN
	THIS^.M_SetError(100, 'Abort button pressed!');
	bAbort := TRUE;

END_IF
END_METHOD

(* Runs for a single cycle when exiting the idle state. *)
METHOD M212_Idle_Exit : BOOL
END_METHOD

(* Runs for a single cycle when entering the starting state. *)
METHOD M300_Starting_Entry : BOOL
THIS^.M_LogMessage('Starting');

// Reset device status variables
bDeviceProgramLoaded := FALSE;
bDevicePoweredOn := FALSE;
bDeviceEnabled := FALSE;
bDeviceProgramStarted := FALSE;
END_METHOD

(* This state should make any final preparations needed for the 'Execute' state
prior to entering the 'Execute' state. *)
METHOD M301_Starting : BOOL
VAR_OUTPUT
	(* This should be set to true once the module and its components are fully
	prepared for process execution. Once set to true, the state machine will
	move to the 'Execute' state. *)
	bStarted	: BOOL;
	(* This should be set to true if an external source requests that the module
	exit its current state and come to a controlled stop. Once set to true, the
	state machine will move to the 'Stopping' state. *)
	bStop	: BOOL;
	(* This should be set to true if a potentially hazardous error or a safety
	fault has occurred in any tasks. Once set to true, the state machine will
	move to the 'Aborting' state. *)
	bAbort	: BOOL;
END_VAR
// Stop if stop button is pressed
bStop := in_bStopBtn;

// Load a program on the device
IF NOT bDeviceProgramLoaded THEN
	bDeviceProgramLoaded := ref_fbDevice.M_LoadProgram(in_strProgram);

// Power on the device
ELSIF NOT bDevicePoweredOn THEN
	bDevicePoweredOn := ref_fbDevice.M_PowerOn();

// Enable the device
ELSIF NOT bDeviceEnabled THEN
	bDeviceEnabled := ref_fbDevice.M_Enable();
	
// Start the device program
ELSIF NOT bDeviceProgramStarted THEN
	bDeviceProgramStarted := ref_fbDevice.M_StartProgram();

// Go to execute state once device program is started
ELSE
	bStarted := TRUE;
END_IF

// If the device has an error, abort
IF ref_fbDevice.P_bError THEN
	THIS^.M_SetError(200, 'Error on fbDevice!');
	bAbort := TRUE;
	
// Abort if abort button is pressed
ELSIF in_bAbortBtn THEN
	THIS^.M_SetError(100, 'Abort button pressed!');
	bAbort := TRUE;

END_IF
END_METHOD

(* Runs for a single cycle when exiting the starting state. *)
METHOD M302_Starting_Exit : BOOL
END_METHOD

(* Runs for a single cycle when entering the execute state. *)
METHOD M310_Execute_Entry : BOOL
THIS^.M_LogMessage('Execute');
END_METHOD

(* The module should remain in this state while it is actively performing
automated tasks. Once all work is finished the state machine should move to the
'Completing' state. *)
METHOD M311_Execute : BOOL
VAR_OUTPUT
	(* This should be set to true once all tasks are complete and automated
	execution should be ended. Once set to true, the state machine will move to
	the 'Completing' state. *)
	bFinished	: BOOL;
	(* This should be set to true as a result of an explicit 'Hold' command
	or if internal conditions require the module to stop operation without
	completely exiting the execution sequence. Once set to true, the state
	machine will move to the 'Holding' state. *)
	bHold	: BOOL;
	(* This should be set to true if external conditions require the module to
	suspend operation until the external conditions are cleared. Once set to
	true, the state machine will move to the 'Suspending' state. *)
	bSuspend	: BOOL;
	(* This should be set to true if an external source requests that the module
	exit its current state and come to a controlled stop. Once set to true, the
	state machine will move to the 'Stopping' state. *)
	bStop	: BOOL;
	(* This should be set to true if a potentially hazardous error or a safety
	fault has occurred in any tasks. Once set to true, the state machine will
	move to the 'Aborting' state. *)
	bAbort	: BOOL;
END_VAR
// Complete if the complete button is pressed
bFinished := in_bCompleteBtn;

// Hold if the hold button is pressed
bHold := in_bHoldBtn;

// Suspend if the suspend button is pressed
bSuspend := in_bSuspendBtn;

// Stop if the stop button is pressed
bStop := in_bStopBtn;

// If the device has an error, abort
IF ref_fbDevice.P_bError THEN
	THIS^.M_SetError(200, 'Error on fbDevice!');
	bAbort := TRUE;
	
// Abort if abort button is pressed
ELSIF in_bAbortBtn THEN
	THIS^.M_SetError(100, 'Abort button pressed!');
	bAbort := TRUE;
END_IF
END_METHOD

(* Runs for a single cycle when exiting the execute state. *)
METHOD M312_Execute_Exit : BOOL
END_METHOD

(* Runs for a single cycle when entering the completing state. *)
METHOD M320_Completing_Entry : BOOL
THIS^.M_LogMessage('Completing');

// Reset device status variables
bDeviceProgramStopped := FALSE;
bDeviceDisabled := FALSE;
END_METHOD

(* This state will perform any post-execution tasks prior to moving to the
'Completed' state. *)
METHOD M321_Completing : BOOL
VAR_OUTPUT
	(* Move to the Complete state*)
	bCompleted	: BOOL;
	(* This should be set to true if an external source requests that the module
	exit its current state and come to a controlled stop. Once set to true, the
	state machine will move to the 'Stopping' state. *)
	bStop	: BOOL;
	(* This should be set to true if a potentially hazardous error or a safety
	fault has occurred in any tasks. Once set to true, the state machine will
	move to the 'Aborting' state. *)
	bAbort	: BOOL;
END_VAR
// Stop the program on the device
IF NOT bDeviceProgramStopped THEN
	bDeviceProgramStopped := ref_fbDevice.M_StopProgram();
	
// Disable the device
ELSIF NOT bDeviceDisabled THEN
	bDeviceDisabled := ref_fbDevice.M_Disable();
	
// Once stoppe and disabled, execution is complete
ELSE
	bCompleted := TRUE;
END_IF

// Stop if the stop button is pressed
bStop := in_bStopBtn;

// If the device has an error, abort
IF ref_fbDevice.P_bError THEN
	THIS^.M_SetError(200, 'Error on fbDevice!');
	bAbort := TRUE;
	
// Abort if abort button is pressed
ELSIF in_bAbortBtn THEN
	THIS^.M_SetError(100, 'Abort button pressed!');
	bAbort := TRUE;
END_IF
END_METHOD

(* Runs for a single cycle when exiting the completing state. *)
METHOD M322_Completing_Exit : BOOL
END_METHOD

(* Runs for a single cycle when entering the complete state. *)
METHOD M330_Complete_Entry : BOOL
THIS^.M_LogMessage('Complete');
END_METHOD

(* The module should remain stationary within this state while maintaing any
execution statistics and awaiting an explicit 'Return' command. *)
METHOD M331_Complete : BOOL
VAR_OUTPUT
	(* This should be set to true if an explicit 'Return' command is received.
	Once set to true, the state machine will move to the 'Resetting' state. *)
	bReturn	: BOOL;
	(* This should be set to true if an external source requests that the module
	exit its current state and come to a controlled stop. Once set to true, the
	state machine will move to the 'Stopping' state. *)
	bStop	: BOOL;
	(* This should be set to true if a potentially hazardous error or a safety
	fault has occurred in any tasks. Once set to true, the state machine will
	move to the 'Aborting' state. *)
	bAbort	: BOOL;
END_VAR
// Return if the reset button is pressed
bReturn := in_bResetBtn;

// Stop if the stop button is pressed
bStop := in_bStopBtn;

// If the device has an error, abort
IF ref_fbDevice.P_bError THEN
	THIS^.M_SetError(200, 'Error on fbDevice!');
	bAbort := TRUE;
	
// Abort if abort button is pressed
ELSIF in_bAbortBtn THEN
	THIS^.M_SetError(100, 'Abort button pressed!');
	bAbort := TRUE;
END_IF
END_METHOD

(* Runs for a single cycle when exiting the complete state. *)
METHOD M332_Complete_Exit : BOOL
END_METHOD

(* Runs for a single cycle when entering the holding state. *)
METHOD M400_Holding_Entry : BOOL
THIS^.M_LogMessage('Holding');

// Reset device state variables
bDeviceProgramPaused := FALSE;
END_METHOD

(* This state should safely pause task executions without completely ending or
resetting them. *)
METHOD M401_Holding : BOOL
VAR_OUTPUT
	(* This should be set to true once all execution tasks are safely paused.
	Once set to true, the state machine will move to the 'Held' state. *)
	bHeld	: BOOL;
	(* This should be set to true if an external source requests that the module
	exit its current state and come to a controlled stop. Once set to true, the
	state machine will move to the 'Stopping' state. *)
	bStop	: BOOL;
	(* This should be set to true if a potentially hazardous error or a safety
	fault has occurred in any tasks. Once set to true, the state machine will
	move to the 'Aborting' state. *)
	bAbort	: BOOL;
END_VAR
// Pause the device
IF NOT bDeviceProgramPaused THEN
	bDeviceProgramPaused := ref_fbDevice.M_PauseProgram();
	
// Once the device is paused, done holding
ELSE
	bHeld := TRUE;
END_IF

// Stop if the stop button is pressed
bStop := in_bStopBtn;

// If the device has an error, abort
IF ref_fbDevice.P_bError THEN
	THIS^.M_SetError(200, 'Error on fbDevice!');
	bAbort := TRUE;
	
// Abort if abort button is pressed
ELSIF in_bAbortBtn THEN
	THIS^.M_SetError(100, 'Abort button pressed!');
	bAbort := TRUE;
END_IF
END_METHOD

(* Runs for a single cycle when exiting the holding state. *)
METHOD M402_Holding_Exit : BOOL
END_METHOD

(* Runs for a single cycle when entering the held state. *)
METHOD M410_Held_Entry : BOOL
THIS^.M_LogMessage('Held');
END_METHOD

(* In this state the most recent execution status should be maintained while
awaiting an explicit 'Unhold' command once internal conditions are satisfactory. *)
METHOD M411_Held : BOOL
VAR_OUTPUT
	(* This should be set to true if an explicit 'Unhold' command is received.
	Once set to true, the state machine will move to the 'Unholding' state. *)
	bUnhold	: BOOL;
	(* This should be set to true if an external source requests that the module
	exit its current state and come to a controlled stop. Once set to true, the
	state machine will move to the 'Stopping' state. *)
	bStop	: BOOL;
	(* This should be set to true if a potentially hazardous error or a safety
	fault has occurred in any tasks. Once set to true, the state machine will
	move to the 'Aborting' state. *)
	bAbort	: BOOL;
END_VAR
// Unhold if the start button is pressed
bUnhold := in_bStartBtn;

// Stop if the stop button is pressed
bStop := in_bStopBtn;

// If the device has an error, abort
IF ref_fbDevice.P_bError THEN
	THIS^.M_SetError(200, 'Error on fbDevice!');
	bAbort := TRUE;
	
// Abort if abort button is pressed
ELSIF in_bAbortBtn THEN
	THIS^.M_SetError(100, 'Abort button pressed!');
	bAbort := TRUE;
END_IF
END_METHOD

(* Runs for a single cycle when exiting the held state. *)
METHOD M412_Held_Exit : BOOL
END_METHOD

(* Runs for a single cycle when entering the unholding state. *)
METHOD M420_Unholding_Entry : BOOL
THIS^.M_LogMessage('Unholding');

// Reset device status variables
bDeviceProgramStarted := FALSE;
END_METHOD

(* In this state, the module and its components should be returned to the
scenario it was in before it entered the 'Holding' step so that the
'Execute' state can pick up where it left off. *)
METHOD M421_Unholding : BOOL
VAR_OUTPUT
	(* This should be set to true once the module is ready to restart
	execution. Once set to true, the state machine will move to the 'Execute'
	state. *)
	bUnheld	: BOOL;
	(* This should be set to true if an external source requests that the module
	exit its current state and come to a controlled stop. Once set to true, the
	state machine will move to the 'Stopping' state. *)
	bStop	: BOOL;
	(* This should be set to true if a potentially hazardous error or a safety
	fault has occurred in any tasks. Once set to true, the state machine will
	move to the 'Aborting' state. *)
	bAbort	: BOOL;
END_VAR
// Restart the device program
IF NOT bDeviceProgramStarted THEN
	bDeviceProgramStarted := ref_fbDevice.M_StartProgram();

// Once the program is started, unholding is finished
ELSE
	bUnheld := TRUE;
END_IF

// Stop if the stop button is pressed
bStop := in_bStopBtn;

// If the device has an error, abort
IF ref_fbDevice.P_bError THEN
	THIS^.M_SetError(200, 'Error on fbDevice!');
	bAbort := TRUE;
	
// Abort if abort button is pressed
ELSIF in_bAbortBtn THEN
	THIS^.M_SetError(100, 'Abort button pressed!');
	bAbort := TRUE;
END_IF
END_METHOD

(* Runs for a single cycle when exiting the unholding state. *)
METHOD M422_Unholding_Exit : BOOL
END_METHOD

(* Runs for a single cycle when entering the suspending state. *)
METHOD M500_Suspending_Entry : BOOL
THIS^.M_LogMessage('Suspending');

// Reset device state variables
bDeviceProgramPaused := FALSE;
END_METHOD

(* This state should safely pause task executions without completely ending or
resetting them. *)
METHOD M501_Suspending : BOOL
VAR_OUTPUT
	(* This should be set to true once all execution tasks are safely paused.
	Once set to true, the state machine will move to the 'Suspended' state. *)
	bSuspended	: BOOL;
	(* This should be set to true if an external source requests that the module
	exit its current state and come to a controlled stop. Once set to true, the
	state machine will move to the 'Stopping' state. *)
	bStop	: BOOL;
	(* This should be set to true if a potentially hazardous error or a safety
	fault has occurred in any tasks. Once set to true, the state machine will
	move to the 'Aborting' state. *)
	bAbort	: BOOL;
END_VAR
// Pause the device
IF NOT bDeviceProgramPaused THEN
	bDeviceProgramPaused := ref_fbDevice.M_PauseProgram();
	
// Once the device is paused, done suspending
ELSE
	bSuspended := TRUE;
END_IF

// Stop if the stop button is pressed
bStop := in_bStopBtn;

// If the device has an error, abort
IF ref_fbDevice.P_bError THEN
	THIS^.M_SetError(200, 'Error on fbDevice!');
	bAbort := TRUE;
	
// Abort if abort button is pressed
ELSIF in_bAbortBtn THEN
	THIS^.M_SetError(100, 'Abort button pressed!');
	bAbort := TRUE;
END_IF
END_METHOD

(* Runs for a single cycle when exiting the suspending state. *)
METHOD M502_Suspending_Exit : BOOL
END_METHOD

(* Runs for a single cycle when entering the suspended state. *)
METHOD M510_Suspended_Entry : BOOL
THIS^.M_LogMessage('Suspended');
END_METHOD

(* In this state the most recent execution status should be maintained while
awaiting an explicit 'Unsuspend' command once external conditions are satisfactory. *)
METHOD M511_Suspended : BOOL
VAR_OUTPUT
	(* This should be set to true if an explicit 'Unsuspend' command is received.
	Once set to true, the state machine will move to the 'Unsuspending' state. *)
	bUnsuspend	: BOOL;
	(* This should be set to true if an external source requests that the module
	exit its current state and come to a controlled stop. Once set to true, the
	state machine will move to the 'Stopping' state. *)
	bStop	: BOOL;
	(* This should be set to true if a potentially hazardous error or a safety
	fault has occurred in any tasks. Once set to true, the state machine will
	move to the 'Aborting' state. *)
	bAbort	: BOOL;
END_VAR
// Unsuspend if the start button is pressed
bUnsuspend := in_bStartBtn;

// Stop if the stop button is pressed
bStop := in_bStopBtn;

// If the device has an error, abort
IF ref_fbDevice.P_bError THEN
	THIS^.M_SetError(200, 'Error on fbDevice!');
	bAbort := TRUE;
	
// Abort if abort button is pressed
ELSIF in_bAbortBtn THEN
	THIS^.M_SetError(100, 'Abort button pressed!');
	bAbort := TRUE;
END_IF
END_METHOD

(* Runs for a single cycle when exiting the suspended state. *)
METHOD M512_Suspended_Exit : BOOL
END_METHOD

(* Runs for a single cycle when entering the unsuspending state. *)
METHOD M520_Unsuspending_Entry : BOOL
THIS^.M_LogMessage('Unsuspending');

// Reset device status variables
bDeviceProgramStarted := FALSE;
END_METHOD

(* In this state, the module and its components should be returned to the
scenario it was in before it entered the 'Suspending' step so that the
'Execute' state can pick up where it left off. *)
METHOD M521_Unsuspending : BOOL
VAR_OUTPUT
	(* This should be set to true once the module is ready to restart
	execution. Once set to true, the state machine will move to the 'Execute'
	state. *)
	bUnsuspended	: BOOL;
	(* This should be set to true if an external source requests that the module
	exit its current state and come to a controlled stop. Once set to true, the
	state machine will move to the 'Stopping' state. *)
	bStop	: BOOL;
	(* This should be set to true if a potentially hazardous error or a safety
	fault has occurred in any tasks. Once set to true, the state machine will
	move to the 'Aborting' state. *)
	bAbort	: BOOL;
END_VAR
// Restart the device program
IF NOT bDeviceProgramStarted THEN
	bDeviceProgramStarted := ref_fbDevice.M_StartProgram();

// Once the program is started, unsuspending is finished
ELSE
	bUnsuspended := TRUE;
END_IF

// Stop if the stop button is pressed
bStop := in_bStopBtn;

// If the device has an error, abort
IF ref_fbDevice.P_bError THEN
	THIS^.M_SetError(200, 'Error on fbDevice!');
	bAbort := TRUE;
	
// Abort if abort button is pressed
ELSIF in_bAbortBtn THEN
	THIS^.M_SetError(100, 'Abort button pressed!');
	bAbort := TRUE;
END_IF
END_METHOD

(* Runs for a single cycle when exiting the unsuspending state. *)
METHOD M522_Unsuspending_Exit : BOOL
END_METHOD

ACTION A_DeviceTestTracking:
// Check device error state
fbDeviceAborted(CLK:=ref_fbDevice.P_bError);
fbDeviceReset(CLK:=ref_fbDevice.P_bError);

// Check device connection state
fbDeviceConnected(CLK:=ref_fbDevice.P_bConnected);
fbDeviceDisconnected(CLK:=ref_fbDevice.P_bConnected);

// Check device enable state
fbDeviceEnabled(CLK:=ref_fbDevice.P_bEnabled);
fbDeviceDisabled(CLK:=ref_fbDevice.P_bEnabled);

// Check device power state
fbDevicePoweredOn(CLK:=ref_fbDevice.P_bPoweredOn);
fbDevicePoweredOff(CLK:=ref_fbDevice.P_bPoweredOn);

// Check device program load state
fbDeviceProgramLoaded(CLK:=(
	ref_fbDevice.P_strCurrentProgram = in_strProgram
	AND LEN(in_strProgram) > 0));
	
// Set outputs based on triggers
IF fbDeviceAborted.Q		THEN out_bAbortTested 		:= TRUE; END_IF
IF fbDeviceReset.Q			THEN out_bResetTested 		:= TRUE; END_IF
IF fbDeviceConnected.Q		THEN out_bConnectTested 	:= TRUE; END_IF
IF fbDeviceDisconnected.Q	THEN out_bDisconnectTested	:= TRUE; END_IF
IF fbDeviceEnabled.Q		THEN out_bEnableTested 		:= TRUE; END_IF
IF fbDeviceDisabled.Q		THEN out_bDisableTested 	:= TRUE; END_IF
IF fbDevicePoweredOn.Q		THEN out_bPowerOnTested 	:= TRUE; END_IF
IF fbDevicePoweredOff.Q		THEN out_bPowerOffTested 	:= TRUE; END_IF
IF fbDeviceProgramLoaded.Q	THEN out_bLoadProgramTested	:= TRUE; END_IF

// Set program control state outputs
IF enumLastState = E_ProgramState.Stopped THEN
	IF ref_fbDevice.P_enumProgramState = E_ProgramState.Running THEN
		out_bStartProgramTested := TRUE;
	END_IF
ELSIF enumLastState = E_ProgramState.Running THEN
	IF ref_fbDevice.P_enumProgramState = E_ProgramState.Stopped THEN
		out_bStopProgramTested := TRUE;
	ELSIF ref_fbDevice.P_enumProgramState = E_ProgramState.Paused THEN
		out_bPauseProgramTested := TRUE;
	END_IF
ELSIF enumLastState = E_ProgramState.Paused THEN
	IF ref_fbDevice.P_enumProgramState = E_ProgramState.Running THEN
		out_bUnpauseProgramTested := TRUE;
	ELSIF ref_fbDevice.P_enumProgramState = E_ProgramState.Stopped THEN
		out_bStopPausedProgramTested := TRUE;
	END_IF
END_IF
enumLastState := ref_fbDevice.P_enumProgramState;
END_ACTION

END_FUNCTION_BLOCK

// Concrete/FB_SimpleMachine
(*
	Machine function block for the Gigavac High Volume FFT machines
*)
{attribute 'hide_all_locals'}
FUNCTION_BLOCK FB_SimpleMachine EXTENDS FB_Machine IMPLEMENTS I_SimpleWaitingStatesOnly
VAR_INPUT
	(* Immediately abort all stations from whatever state they are in and
		go to the Aborted state. *)
	in_bAbortBtn : BOOL;
	(* Immediately stop all stations from whatever state they are in and
		go to the Stopped state. *)
	in_bStopBtn : BOOL;
	(* Clear all stations from the Aborted state and go to the Stopped state. *)
	in_bClearBtn : BOOL;
	(* Reset all stations from the Stopped state and go to the Idle state. *)
	in_bResetBtn : BOOL;
	(* Start all stations from the Idle state and go to the Execute state. *)
	in_bStartBtn : BOOL;
	(* Hold all stations from the Execute state and go to the Held state. *)
	in_bHoldBtn : BOOL;
	(* Unhold all stations from the Held state and go to the Execute state. *)
	in_bUnholdBtn : BOOL;
	(* Suspend all stations from the Execute state and go to the Held Suspended. *)
	in_bSuspendBtn : BOOL;
	(* Unsuspend all stations from the Suspended state and go to the Execute state. *)
	in_bUnsuspendBtn : BOOL;
	(* Complete all stations from the Execute state and go to the Completed state. *)
	in_bCompleteBtn : BOOL;
	(* Return all stations from the Completed state and go to the Idle state. *)
	in_bReturnBtn : BOOL;
END_VAR
VAR_OUTPUT
END_VAR
VAR
	// Abort
	smac_fbAbortTrig: R_TRIG;
	smac_bAbortTrig: BOOL;
	smac_bAborting: BOOL;
	smac_bAborted: BOOL;

	// Stop
	smac_fbStopTrig: R_TRIG;
	smac_bStopTrig: BOOL;
	smac_bStopping: BOOL;
	smac_bStopped: BOOL;
	
	// Aborted
	smac_fbClearTrig: R_TRIG;
	smac_bClearTrig: BOOL;
	
	// Stopped
	smac_fbResetTrig: R_TRIG;
	smac_bResetTrig: BOOL;
	
	// Idle
	smac_fbStartTrig: R_TRIG;
	smac_bStartTrig: BOOL;
	
	// Execute
	smac_fbCompleteTrig: R_TRIG;
	smac_bCompleteTrig: BOOL;
	smac_fbHoldTrig: R_TRIG;
	smac_bHoldTrig: BOOL;
	smac_fbSuspendTrig: R_TRIG;
	smac_bSuspendTrig: BOOL;
	
	// Complete
	smac_fbReturnTrig: R_TRIG;
	smac_bReturnTrig: BOOL;
	
	// Held
	smac_fbUnholdTrig: R_TRIG;
	smac_bUnholdTrig: BOOL;
	
	// Suspended
	smac_fbUnsuspendTrig: R_TRIG;
	smac_bUnsuspendTrig: BOOL;
END_VAR

ACTION A_Buttons:
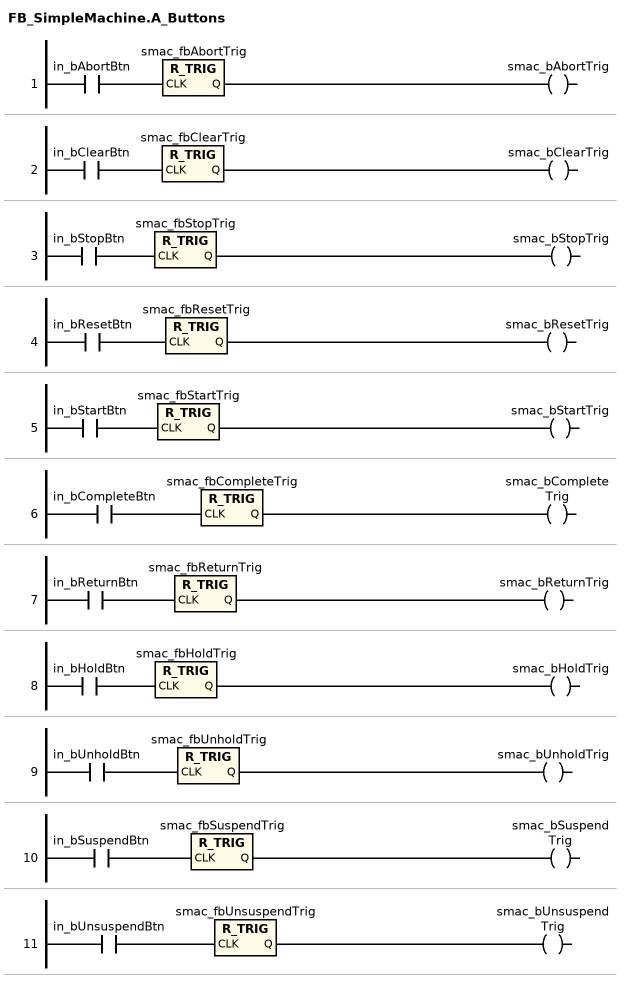
// NETWORK 1
smac_fbAbortTrig(CLK := in_bAbortBtn); // R_TRIG
smac_bAbortTrig := smac_fbAbortTrig.Q;

// NETWORK 2
smac_fbClearTrig(CLK := in_bClearBtn); // R_TRIG
smac_bClearTrig := smac_fbClearTrig.Q;

// NETWORK 3
smac_fbStopTrig(CLK := in_bStopBtn); // R_TRIG
smac_bStopTrig := smac_fbStopTrig.Q;

// NETWORK 4
smac_fbResetTrig(CLK := in_bResetBtn); // R_TRIG
smac_bResetTrig := smac_fbResetTrig.Q;

// NETWORK 5
smac_fbStartTrig(CLK := in_bStartBtn); // R_TRIG
smac_bStartTrig := smac_fbStartTrig.Q;

// NETWORK 6
smac_fbCompleteTrig(CLK := in_bCompleteBtn); // R_TRIG
smac_bCompleteTrig := smac_fbCompleteTrig.Q;

// NETWORK 7
smac_fbReturnTrig(CLK := in_bReturnBtn); // R_TRIG
smac_bReturnTrig := smac_fbReturnTrig.Q;

// NETWORK 8
smac_fbHoldTrig(CLK := in_bHoldBtn); // R_TRIG
smac_bHoldTrig := smac_fbHoldTrig.Q;

// NETWORK 9
smac_fbUnholdTrig(CLK := in_bUnholdBtn); // R_TRIG
smac_bUnholdTrig := smac_fbUnholdTrig.Q;

// NETWORK 10
smac_fbSuspendTrig(CLK := in_bSuspendBtn); // R_TRIG
smac_bSuspendTrig := smac_fbSuspendTrig.Q;

// NETWORK 11
smac_fbUnsuspendTrig(CLK := in_bUnsuspendBtn); // R_TRIG
smac_bUnsuspendTrig := smac_fbUnsuspendTrig.Q;
END_ACTION

ACTION A_RunSimpleMachine:
THIS^.A_StopAndAbort();
THIS^.A_Buttons();
THIS^.A_StateMachine();
END_ACTION

ACTION A_StopAndAbort:
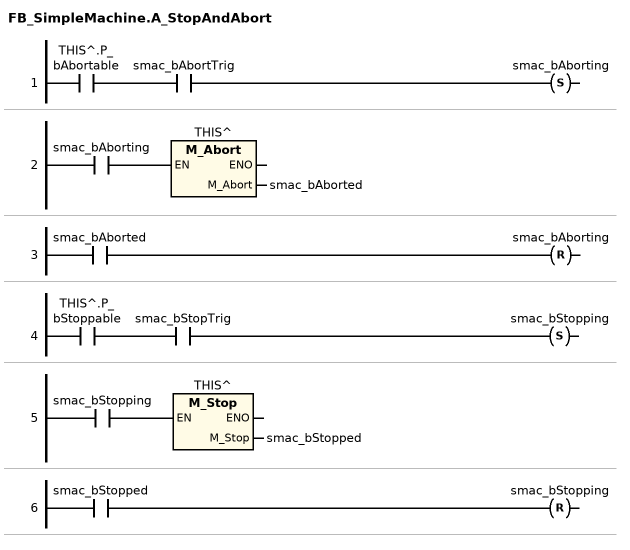
// NETWORK 1
smac_bAborting S= THIS^.P_bAbortable AND smac_bAbortTrig;

// NETWORK 2
IF smac_bAborting THEN THIS^.M_Abort(M_Abort => smac_bAborted); END_IF

// NETWORK 3
smac_bAborting R= smac_bAborted;

// NETWORK 4
smac_bStopping S= THIS^.P_bStoppable AND smac_bStopTrig;

// NETWORK 5
IF smac_bStopping THEN THIS^.M_Stop(M_Stop => smac_bStopped); END_IF

// NETWORK 6
smac_bStopping R= smac_bStopped;
END_ACTION

(* This state is entered after the aborting state completes, and should
not modify anything in the module while awaiting an explicit 'Clear' command. *)
METHOD M011_Aborted : BOOL
VAR_OUTPUT
	(* This should be set to true once an explicit 'Clear' command is received.
	Once set to true, the state machine will move to the 'Clearing' state. *)
	bClear	: BOOL;
END_VAR
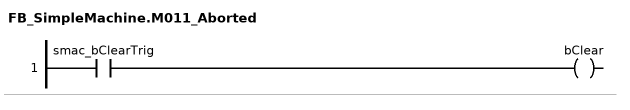
// NETWORK 1
bClear := smac_bClearTrig;
END_METHOD

(* The machine should be stationary and awaiting an explicit 'Reset' command
while in this state. Once the 'Reset' command is received, the state machine
will move to the 'Resetting' state. *)
METHOD M111_Stopped : BOOL
VAR_OUTPUT
	(* This should be set to true if an explicit reset command is received.
	Once set to true, the state machine will move to the 'Resetting' state. *)
	bReset	: BOOL;
	(* This should be set to true if a potentially hazardous error or a safety
	fault has occurred in any tasks. Once set to true, the state machine will
	move to the 'Aborting' state. *)
	bAbort	: BOOL;
END_VAR
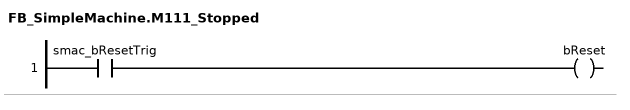
// NETWORK 1
bReset := smac_bResetTrig;
END_METHOD

(* This state should maintain the status of the module and its components that
was set by the resetting step while awaiting an explicit 'Start' command. *)
METHOD M211_Idle : BOOL
VAR_OUTPUT
	(* This should be set to true if an explicit 'Start' command is received.
	Once set to true, the state machine will move to the 'Starting' state. *)
	bStart	: BOOL;
	(* This should be set to true if an external source requests that the module
	exit its current state and come to a controlled stop. Once set to true, the
	state machine will move to the 'Stopping' state. *)
	bStop	: BOOL;
	(* This should be set to true if a potentially hazardous error or a safety
	fault has occurred in any tasks. Once set to true, the state machine will
	move to the 'Aborting' state. *)
	bAbort	: BOOL;
END_VAR
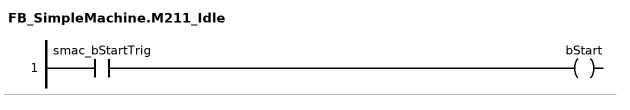
// NETWORK 1
bStart := smac_bStartTrig;
END_METHOD

(* The module should remain in this state while it is actively performing
automated tasks. Once all work is finished the state machine should move to the
'Completing' state. *)
METHOD M311_Execute : BOOL
VAR_OUTPUT
	(* This should be set to true once all tasks are complete and automated
	execution should be ended. Once set to true, the state machine will move to
	the 'Completing' state. *)
	bFinished	: BOOL;
	(* This should be set to true as a result of an explicit 'Hold' command
	or if internal conditions require the module to stop operation without
	completely exiting the execution sequence. Once set to true, the state
	machine will move to the 'Holding' state. *)
	bHold	: BOOL;
	(* This should be set to true if external conditions require the module to
	suspend operation until the external conditions are cleared. Once set to
	true, the state machine will move to the 'Suspending' state. *)
	bSuspend	: BOOL;
	(* This should be set to true if an external source requests that the module
	exit its current state and come to a controlled stop. Once set to true, the
	state machine will move to the 'Stopping' state. *)
	bStop	: BOOL;
	(* This should be set to true if a potentially hazardous error or a safety
	fault has occurred in any tasks. Once set to true, the state machine will
	move to the 'Aborting' state. *)
	bAbort	: BOOL;
END_VAR
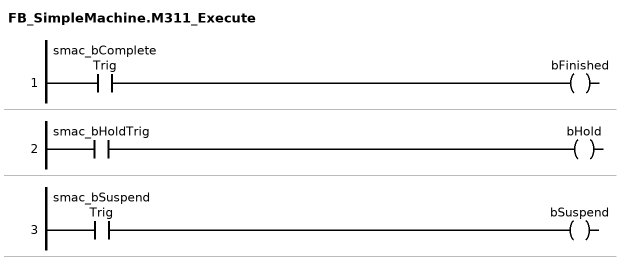
// NETWORK 1
bFinished := smac_bCompleteTrig;

// NETWORK 2
bHold := smac_bHoldTrig;

// NETWORK 3
bSuspend := smac_bSuspendTrig;
END_METHOD

(* The module should remain stationary within this state while maintaing any
execution statistics and awaiting an explicit 'Return' command. *)
METHOD M331_Complete : BOOL
VAR_OUTPUT
	(* This should be set to true if an explicit 'Return' command is received.
	Once set to true, the state machine will move to the 'Resetting' state. *)
	bReturn	: BOOL;
	(* This should be set to true if an external source requests that the module
	exit its current state and come to a controlled stop. Once set to true, the
	state machine will move to the 'Stopping' state. *)
	bStop	: BOOL;
	(* This should be set to true if a potentially hazardous error or a safety
	fault has occurred in any tasks. Once set to true, the state machine will
	move to the 'Aborting' state. *)
	bAbort	: BOOL;
END_VAR
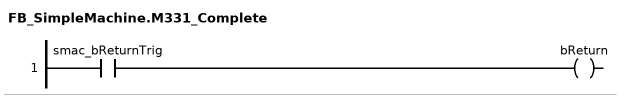
// NETWORK 1
bReturn := smac_bReturnTrig;
END_METHOD

(* In this state the most recent execution status should be maintained while
awaiting an explicit 'Unhold' command once internal conditions are satisfactory. *)
METHOD M411_Held : BOOL
VAR_OUTPUT
	(* This should be set to true if an explicit 'Unhold' command is received.
	Once set to true, the state machine will move to the 'Unholding' state. *)
	bUnhold	: BOOL;
	(* This should be set to true if an external source requests that the module
	exit its current state and come to a controlled stop. Once set to true, the
	state machine will move to the 'Stopping' state. *)
	bStop	: BOOL;
	(* This should be set to true if a potentially hazardous error or a safety
	fault has occurred in any tasks. Once set to true, the state machine will
	move to the 'Aborting' state. *)
	bAbort	: BOOL;
END_VAR
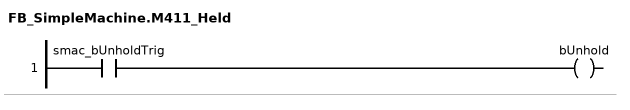
// NETWORK 1
bUnhold := smac_bUnholdTrig;
END_METHOD

(* In this state the most recent execution status should be maintained while
awaiting an explicit 'Unsuspend' command once external conditions are satisfactory. *)
METHOD M511_Suspended : BOOL
VAR_OUTPUT
	(* This should be set to true if an explicit 'Unsuspend' command is received.
	Once set to true, the state machine will move to the 'Unsuspending' state. *)
	bUnsuspend	: BOOL;
	(* This should be set to true if an external source requests that the module
	exit its current state and come to a controlled stop. Once set to true, the
	state machine will move to the 'Stopping' state. *)
	bStop	: BOOL;
	(* This should be set to true if a potentially hazardous error or a safety
	fault has occurred in any tasks. Once set to true, the state machine will
	move to the 'Aborting' state. *)
	bAbort	: BOOL;
END_VAR
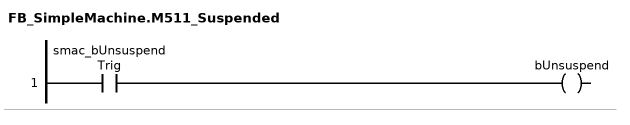
// NETWORK 1
bUnsuspend := smac_bUnsuspendTrig;
END_METHOD

END_FUNCTION_BLOCK

// Interfaces/State Machine/Stateful/I_ExecuteStateOnly
(* This interface only implements the methods for the Execute state. *)
INTERFACE I_ExecuteStateOnly EXTENDS I_SimpleExecuteStateOnly

(* Runs for a single cycle when entering the execute state. *)
METHOD M310_Execute_Entry : BOOL
VAR_INPUT
END_VAR
END_METHOD

(* Runs for a single cycle when exiting the execute state. *)
METHOD M312_Execute_Exit : BOOL
VAR_INPUT
END_VAR
END_METHOD

END_INTERFACE

// Interfaces/State Machine/Stateful/I_TransitionStatesOnly
(* This interface implements only the PackML transition states. *)
INTERFACE I_TransitionStatesOnly EXTENDS I_SimpleTransitionStatesOnly

(* Runs for a single cycle when entering the aborting state. *)
METHOD M000_Aborting_Entry : BOOL
VAR_INPUT
END_VAR
END_METHOD

(* Runs for a single cycle when exiting the aborting state. *)
METHOD M002_Aborting_Exit : BOOL
VAR_INPUT
END_VAR
END_METHOD

(* Runs for a single cycle when entering the clearing state. *)
METHOD M020_Clearing_Entry : BOOL
VAR_INPUT
END_VAR
END_METHOD

(* Runs for a single cycle when exiting the clearing state. *)
METHOD M022_Clearing_Exit : BOOL
VAR_INPUT
END_VAR
END_METHOD

(* Runs for a single cycle when entering the stopping state. *)
METHOD M100_Stopping_Entry : BOOL
VAR_INPUT
END_VAR
END_METHOD

(* Runs for a single cycle when exiting the stopping state. *)
METHOD M102_Stopping_Exit : BOOL
VAR_INPUT
END_VAR
END_METHOD

(* Runs for a single cycle when entering the resetting state. *)
METHOD M200_Resetting_Entry : BOOL
VAR_INPUT
END_VAR
END_METHOD

(* Runs for a single cycle when exiting the resetting state. *)
METHOD M202_Resetting_Exit : BOOL
VAR_INPUT
END_VAR
END_METHOD

(* Runs for a single cycle when entering the starting state. *)
METHOD M300_Starting_Entry : BOOL
VAR_INPUT
END_VAR
END_METHOD

(* Runs for a single cycle when exiting the starting state. *)
METHOD M302_Starting_Exit : BOOL
VAR_INPUT
END_VAR
END_METHOD

(* Runs for a single cycle when entering the completing state. *)
METHOD M320_Completing_Entry : BOOL
VAR_INPUT
END_VAR
END_METHOD

(* Runs for a single cycle when exiting the completing state. *)
METHOD M322_Completing_Exit : BOOL
VAR_INPUT
END_VAR
END_METHOD

(* Runs for a single cycle when entering the holding state. *)
METHOD M400_Holding_Entry : BOOL
VAR_INPUT
END_VAR
END_METHOD

(* Runs for a single cycle when exiting the holding state. *)
METHOD M402_Holding_Exit : BOOL
VAR_INPUT
END_VAR
END_METHOD

(* Runs for a single cycle when entering the unholding state. *)
METHOD M420_Unholding_Entry : BOOL
VAR_INPUT
END_VAR
END_METHOD

(* Runs for a single cycle when exiting the unholding state. *)
METHOD M422_Unholding_Exit : BOOL
VAR_INPUT
END_VAR
END_METHOD

(* Runs for a single cycle when entering the suspending state. *)
METHOD M500_Suspending_Entry : BOOL
VAR_INPUT
END_VAR
END_METHOD

(* Runs for a single cycle when exiting the suspending state. *)
METHOD M502_Suspending_Exit : BOOL
VAR_INPUT
END_VAR
END_METHOD

(* Runs for a single cycle when entering the unsuspending state. *)
METHOD M520_Unsuspending_Entry : BOOL
VAR_INPUT
END_VAR
END_METHOD

(* Runs for a single cycle when exiting the unsuspending state. *)
METHOD M522_Unsuspending_Exit : BOOL
VAR_INPUT
END_VAR
END_METHOD

END_INTERFACE

// Project Information/F_GetCompany
// This function has been automatically generated from the project information.
{attribute 'signature_flag' := '1073741824'}
{attribute 'TcGenerated'}
{attribute 'no-analysis'}
FUNCTION F_GetCompany : WSTRING
VAR_INPUT
	
END_VAR

F_GetCompany := "Sensata Technologies";

END_FUNCTION

// Project Information/F_GetTitle
// This function has been automatically generated from the project information.
{attribute 'signature_flag' := '1073741824'}
{attribute 'TcGenerated'}
{attribute 'no-analysis'}
FUNCTION F_GetTitle : WSTRING
VAR_INPUT
	
END_VAR

F_GetTitle := "Sensata_Common";

END_FUNCTION

// Project Information/F_GetVersion
// This function has been automatically generated from the project information.
{attribute 'signature_flag' := '1073741824'}
{attribute 'TcGenerated'}
{attribute 'no-analysis'}
FUNCTION F_GetVersion : ST_LibVersion
VAR_INPUT
	
END_VAR

F_GetVersion.iMajor := 1;
F_GetVersion.iMinor := 0;
F_GetVersion.iBuild := 0;
F_GetVersion.iRevision := 0;

END_FUNCTION
